
FUNCTION CB_real_to_byte : BYTE


TITLE = ' Convert a real into a byte '
VERSION : '1.0'
AUTHOR  : CB
NAME    : realByte
FAMILY  : TNI

VAR_INPUT
    IN : REAL;
END_VAR

VAR_TEMP

END_VAR

BEGIN

CB_real_to_byte :=INT_TO_BYTE(REAL_TO_INT(IN));

END_FUNCTION
